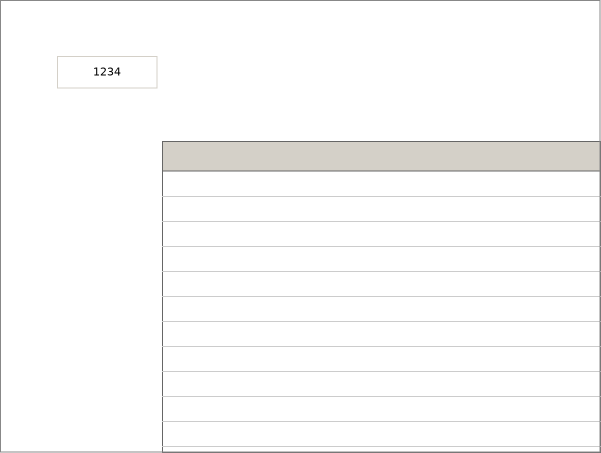
VISUALIZATION visValveControl  // 601x453
    Textfield (57,56 100x32), "1234"
        OnMouseClick: write GVL_visVariableMap.nValveMask via VisuDialogs.Numpad
    Table (162,141 439x312), data array: GVL_visVariableMap.anValveMask
        p3854506369: GVL_visVariableMap.anValveMask[INDEX]
END_VISUALIZATION

(* stored: Version 1.1.0.1
   Visu visValveControl: Id {d66bddad-486a-0fc1-209a-74dad9554183} *)
